{attribute 'qualified_only'}
VAR_GLOBAL
		EtherCAT_Master_ELXxxxx : EtherCAT_Master_ELXxxxx_2690D376;
END_VAR

(* stored: Version 1.2.0.0, ProductVersion 3.1.4024.9
   GVL GVL_iXlinker: Id {2d5bef85-3065-43ee-9083-c923ee89f277} *)
